TYPE
    ST_MotorMonitor :
    STRUCT
        InForward  : BOOL;
        InBackward : BOOL;
        InStopped  : BOOL;
        Error      : BOOL;
        ErrMsg     : T_MaxString;
    END_STRUCT
END_TYPE

(* stored: Version 1.1.0.1, ProductVersion 3.1.4024.13
   DUT ST_MotorMonitor: Id {0e8d077f-a292-4fc7-b201-f46a877c2db8} *)
